PROGRAM MAIN
VAR
END_VAR

END_PROGRAM

(* stored: Version 1.1.0.1
   POU MAIN: Id {9005e2b7-240f-4984-9240-b0acc1618302} *)
